// TwinCAT 3 PLC project Coffee_maker_PLC
// ProgramVersion: 3.1.4024.0
// libraries:
//   Tc2_Standard, * (Beckhoff Automation GmbH)
//   Tc2_System, * (Beckhoff Automation GmbH)
//   Tc3_Module, * (Beckhoff Automation GmbH)
// project tree:
//   / GlobalTextList.TcGTLO, PlcTask.TcTTO, Visualization Manager.TcVMO (not stored)
//   GVLs/ GVL.TcGVL
//   POUs/ Cleaning.TcPOU, Fill_Cup.TcPOU, Heat_Water.TcPOU, Lamp_Loop.TcPOU, MAIN.TcPOU, Prepare_Ingredients.TcPOU, Show_Strength.TcPOU
//   VISUs/ Visualization.TcVIS
// real-time tasks:
//   TASK PlcTask: cycle T#10ms, priority 20, ADS port 350
//   TASK Fill_Cup: cycle T#10ms, priority 1, ADS port 351
//   TASK Prepare_Ingredients: cycle T#5ms, priority 2, ADS port 352
//   TASK Heating: cycle T#1ms, priority 3, ADS port 353
//   TASK LoopLamp: cycle T#10ms, priority 4, ADS port 354
//   TASK Show strength: cycle T#10ms, priority 5, ADS port 355

CONFIGURATION Coffee_maker_PLC
    RESOURCE PLC ON TwinCAT3
        TASK PlcTask(INTERVAL := T#10ms, PRIORITY := 20);
        PROGRAM MAIN WITH PlcTask : MAIN;
        PROGRAM Fill_Cup WITH PlcTask : Fill_Cup;
        PROGRAM Heat_Water WITH PlcTask : Heat_Water;
        PROGRAM Lamp_Loop WITH PlcTask : Lamp_Loop;
        PROGRAM Prepare_Ingredients WITH PlcTask : Prepare_Ingredients;
        PROGRAM Show_Strength WITH PlcTask : Show_Strength;
    END_RESOURCE
END_CONFIGURATION

// ---- GVLs/GVL.TcGVL
{attribute 'qualified_only'}
VAR_GLOBAL
	Start : BOOL := FALSE;	
	CleanMachine : BOOL := FALSE;
	FillCup : BOOL := FALSE;
	Water_Warm: BOOL := FALSE;
    Ingredients_Ready : BOOL := FALSE;
	Cup_filled : BOOL := FALSE;
	Coffee_Strength : INT;
	LamploopOn : BOOL := FALSE;
	Strength : INT := 0;
	Lamp1 : BOOL := FALSE; // Output for Lamp 1
    Lamp2 : BOOL := FALSE; // Output for Lamp 2
    Lamp3 : BOOL := FALSE; // Output for Lamp 3
	ShowStrength : BOOL := FALSE;
END_VAR

// ---- POUs/MAIN.TcPOU
PROGRAM MAIN
VAR
	cleaningfb1: Cleaning;
END_VAR

IF gvl.CleanMachine = TRUE THEN 
	Cleaning(TypeCleaning := 1);
END_IF

END_PROGRAM

// ---- POUs/Cleaning.TcPOU
FUNCTION_BLOCK Cleaning
VAR_INPUT
	TypeCleaning : INT;
END_VAR
VAR_OUTPUT
END_VAR
VAR
	MachineClean : BOOL := FALSE;
	CleaningStep : INT := 0;
	WaitTime : TIME := T#2S; // Stel de wachttijd in voor elke stap
    Timer : TIME := T#0s;
    CleaningDone : BOOL := FALSE;
END_VAR

IF TypeCleaning = 1 THEN 
	// grote schoonmaak 
	// Reset schoonmaak gereed status
	MachineClean := FALSE;
	
	IF NOT CleaningDone THEN
		CASE CleaningStep OF
		0:
			// Stap 1: Begin het schoonmaakproces
			Timer := Timer + T#100MS;
			IF Timer >= WaitTime THEN
				CleaningStep := CleaningStep + 1;
				Timer := T#0S; // Reset de timer
			END_IF

		1:
			// Stap 2: Spoel de koffieresiduen uit
			Timer := Timer + T#100MS;
			IF Timer >= WaitTime THEN
				CleaningStep := CleaningStep + 1;
				Timer := T#0S;
			END_IF

		2:
			// Stap 3: Reinig waterleidingen
			Timer := Timer + T#100MS;
			IF Timer >= WaitTime THEN
				CleaningStep := CleaningStep + 1;
				Timer := T#0S;
			END_IF
	
		3:
			// Stap 4: Reinig koffiedikopvangbak
			Timer := Timer + T#100MS;
			IF Timer >= WaitTime THEN
				CleaningStep := CleaningStep + 1;
				Timer := T#0S;
			END_IF

		4:
			// Stap 5: Reinig externe oppervlakken
			Timer := Timer + T#100MS;
			IF Timer >= WaitTime THEN
				CleaningDone := TRUE;  // Schoonmaak is gereed
			END_IF
		ELSE
		// Schoonmaakproces voltooid, zet de returnwaarde op TRUE
		MachineClean := TRUE;
		END_CASE
	END_IF

	
	
ELSIF TypeCleaning = 2 THEN 
	// kleine reineging 
	// Reset schoonmaak gereed status
	MachineClean := FALSE;
	
	
	
	IF NOT CleaningDone THEN
		CASE CleaningStep OF
			0:
				// Stap 1: Spoel koffieresiduen kort door
				Timer := Timer + T#100MS;
				IF Timer >= WaitTime THEN
					CleaningStep := CleaningStep + 1;
					Timer := T#0S; // Reset de timer
				END_IF
	
			1:
				// Stap 2: Spoel waterleidingen kort door
				Timer := Timer + T#100MS;
				IF Timer >= WaitTime THEN
					CleaningStep := CleaningStep + 1;
					Timer := T#0S;
				END_IF
	
			2:
				// Stap 3: Reinig opvangbak oppervlakkig
				Timer := Timer + T#100MS;
				IF Timer >= WaitTime THEN
					CleaningDone := TRUE;  // Kleine schoonmaak is gereed
				END_IF
		ELSE
			// Schoonmaakproces voltooid, zet de returnwaarde op TRUE
			MachineClean := TRUE;
		END_CASE
	END_IF
END_IF

END_FUNCTION_BLOCK

// ---- POUs/Fill_Cup.TcPOU
PROGRAM Fill_Cup
VAR
	Filling : BOOL := FALSE;
	Timer : Ton;
	Licht : BOOL;
	Medium : BOOL; 
	Sterk : BOOL;	
	cleaningfb: Cleaning;
END_VAR

IF gvl.FillCup THEN 
	IF gvl.Water_Warm = TRUE AND gvl.Ingredients_Ready = TRUE THEN
	Timer(IN := TRUE, PT := T#5S); // 5 seconden timer

		IF gvl.Strength = 0 THEN;
			gvl.LamploopOn := true;		
				IF licht  THEN
				gvl.Strength := 1;
				gvl.LamploopOn := FALSE;
				
				ELSIF medium THEN 
				gvl.Strength := 2;
				gvl.LamploopOn := FALSE;
				
				ELSIF sterk THEN
				gvl.Strength := 3;
				gvl.LamploopOn := FALSE;
				END_IF
		END_IF
	
		IF gvl.Strength > 0 THEN
			Filling := TRUE;
			gvl.ShowStrength := 1;
		END_IF
		
		IF Timer.Q THEN 
			Filling := FALSE;
			gvl.Cup_Filled := TRUE;
		END_IF	
		
		Cleaning(TypeCleaning := 2); // korte reiniging 
		
	END_IF
END_IF

END_PROGRAM

// ---- POUs/Heat_Water.TcPOU
PROGRAM Heat_Water
VAR
	WaterTemp: INT := 20;
	Heating : bool := false;
	ELSIFgvl: INT;
	Timer:TON;
	
END_VAR

IF gvl.Start AND WaterTemp <= 85 THEN
    Timer(IN := TRUE, PT := T#100MS);  
    Heating := TRUE;

    IF Timer.Q THEN 
        WaterTemp := WaterTemp + 1;  // Verhoog de temperatuur met 1 graad per seconde
        Timer(IN := FALSE);          // Reset de timer na een seconde
    END_IF

ELSIF gvl.Start = FALSE THEN
    Heating := FALSE;
    Timer(IN := FALSE);              // Zorg ervoor dat de timer wordt gereset als Start FALSE is

ELSIF WaterTemp >= 85 THEN  
    Heating := FALSE;
    gvl.Water_Warm := TRUE;	
    Timer(IN := FALSE);              // Stop de timer als de gewenste temperatuur is bereikt

END_IF

END_PROGRAM

// ---- POUs/Lamp_Loop.TcPOU
PROGRAM Lamp_Loop
VAR
	Strength : INT;
	Lamp1 : BOOL := FALSE; // Output for Lamp 1
    Lamp2 : BOOL := FALSE; // Output for Lamp 2
    Lamp3 : BOOL := FALSE; // Output for Lamp 3

    tCycleTimer : TON; // Timer for cycle timing
    nCycleStep : INT := 0; // State variable to track which lamp is on 
END_VAR

IF gvl.LamploopOn THEN 
	// Timer instellingen
	tCycleTimer(IN := TRUE, PT := T#0.5S); // De timer is ingesteld op 2 seconden
	
	IF tCycleTimer.Q THEN
		tCycleTimer(IN := FALSE);  // Stop de timer zodra deze is afgelopen
		tCycleTimer(IN := TRUE);   // Reset de timer voor de volgende cyclus
	
		// Volgende stap van de cyclus
		nCycleStep := nCycleStep + 1;
		
		IF nCycleStep > 2 THEN
			nCycleStep := 0; // Reset de cyclus na 3 stappen
		END_IF
	END_IF
	
	// Lamp logica
	CASE nCycleStep OF
		0: // Lamp 1 aan, andere uit
			gvl.Lamp1 := TRUE;
			gvl.Lamp2 := FALSE;
			gvl.Lamp3 := FALSE;
		1: // Lamp 2 aan, andere uit
			gvl.Lamp1 := FALSE;
			gvl.Lamp2 := TRUE;
			gvl.Lamp3 := FALSE;
		2: // Lamp 3 aan, andere uit
			gvl.Lamp1 := FALSE;
			gvl.Lamp2 := FALSE;
			gvl.Lamp3 := TRUE;
	END_CASE
END_IF

END_PROGRAM

// ---- POUs/Prepare_Ingredients.TcPOU
PROGRAM Prepare_Ingredients
VAR
	BoneContainer: REAL := 0;	
	Prepairing : BOOL := FALSE;
	Timer:TON;
END_VAR

Timer(IN := TRUE, PT := T#100MS); 				// 1 seconden timer

IF gvl.Start AND BoneContainer <= 90 THEN
    Timer(IN := TRUE, PT := T#1S);   		// Stel de timer in om elke seconde af te gaan
    Prepairing := TRUE;

    IF Timer.Q THEN
        BoneContainer := BoneContainer + 1;  // Verhoog de inhoud van BoneContainer met 1
        Timer(IN := FALSE);                  // Reset de timer na een seconde
    END_IF

ELSIF BoneContainer >= 90 THEN
    gvl.Ingredients_Ready := TRUE;
    Prepairing := FALSE;
    Timer(IN := FALSE);                      // Stop de timer wanneer BoneContainer vol is

ELSIF gvl.Start = FALSE THEN
    Prepairing := FALSE;
    Timer(IN := FALSE);                      // Reset de timer wanneer Start FALSE is
END_IF

END_PROGRAM

// ---- POUs/Show_Strength.TcPOU
PROGRAM Show_Strength
VAR
END_VAR

IF gvl.ShowStrength = TRUE THEN 
	gvl.lamp1 := 0;
	gvl.Lamp2 := 0;
	gvl.Lamp3 := 0;
	
	IF gvl.Strength = 1 THEN 
		gvl.Lamp1 := 1;
	ELSIF gvl.Strength = 2 THEN 
		gvl.Lamp2 := 1;
	ELSIF gvl.Strength = 3 THEN 
		gvl.Lamp3 := 1;
	END_IF
	gvl.ShowStrength := 0;
	
END_IF

END_PROGRAM

// ---- GlobalTextList.TcGTLO
TEXTLIST GlobalTextList
  313 = 'Cleaning Program'
  896 = 'Filling Cup'
  750 = 'Heating'
  77 = 'Koffie klaar'
  777 = 'Licht          Medium        Sterk'
  759 = 'Prepairing Ingredients'
  169 = 'Start'
  681 = 'Start Cleaning Program'
  172 = 'Watertemperatuur'
END_TEXTLIST

// ---- VISUs/Visualization.TcVIS
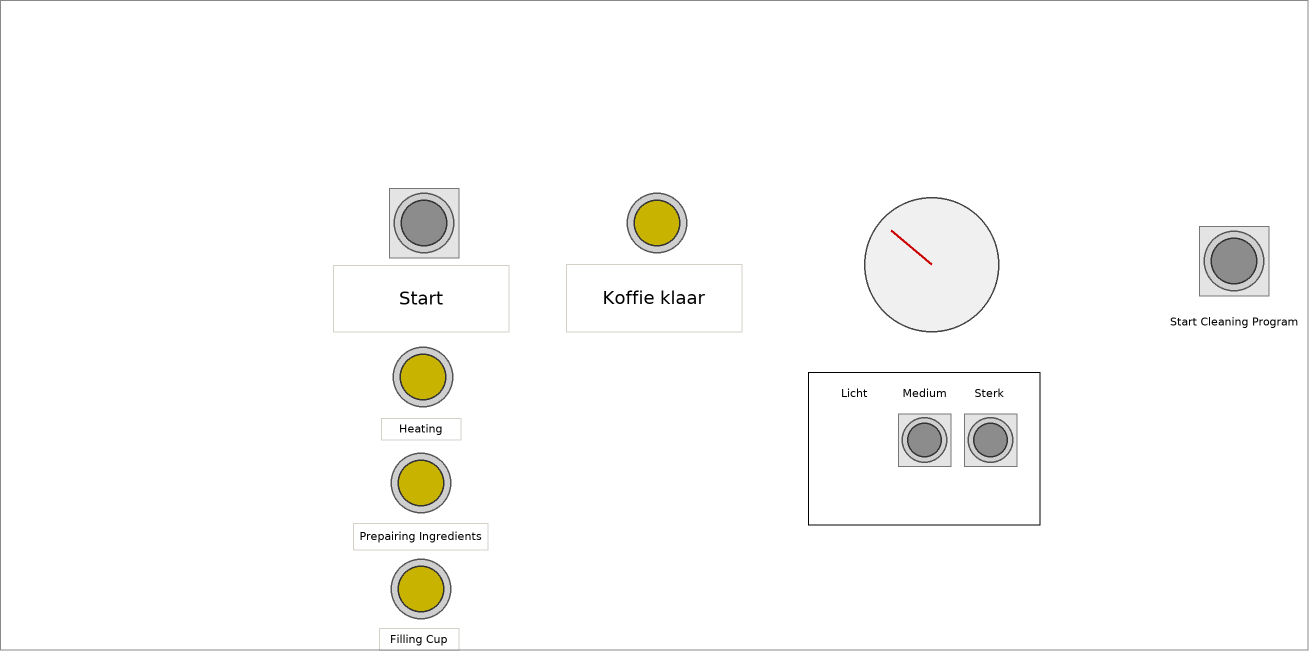
VISUALIZATION Visualization  // 1309x651
    Lamp1 (388,342 70x70), variable: Heating.Heating, style: Lamp-Lamp1-Yellow
    Lamp1 (386,448 70x70), variable: Prepare_Ingredients.Prepairing, style: Lamp-Lamp1-Yellow
    PushSwitchLed (389,188 70x70), variable: GVL.Start, behaviour: TOGGLE, style: Switch-PushSwitchLed-Gray
    Textfield (333,265 176x67), "Start"
    Textfield (381,418 80x22), "Heating"
    Textfield (353,523 135x27), "Prepairing Ingredients"
    Lamp1 (622,188 70x70), variable: Fill_Cup.Ready, style: Lamp-Lamp1-Yellow
    Textfield (566,264 176x68), "Koffie klaar"
    Meter180 (788,197 287x135), value: Heating.WaterTemp, style: Meter-Meter180-Yellow, scale format: %.1f, scale 0..100
        p518627256: Watertemperatuur
    Lamp1 (386,554 70x70), variable: Fill_Cup.Filling, style: Lamp-Lamp1-Yellow
    Textfield (379,628 80x23), "Filling Cup"
    Lamp1 (840,473 41x38), variable: Lamp_Loop.Lamp1, style: Lamp-Lamp1-Yellow
    Lamp1 (907,473 41x38), variable: Lamp_Loop.Lamp2, style: Lamp-Lamp1-Yellow
    Lamp1 (972,473 41x38), variable: Lamp_Loop.Lamp3, style: Lamp-Lamp1-Yellow
    Frame (979,444 1x0)
    PushSwitch (832,410 53x60), variable: Fill_Cup.Licht, behaviour: TOGGLE, style: Switch-PushSwitch-Gray
    Rectangle (808,372 232x153)
    Textfield (813,378 219x31), "Licht Medium Sterk"
    PushSwitch (898,410 53x60), variable: Fill_Cup.Medium, behaviour: TOGGLE, style: Switch-PushSwitch-Gray
    PushSwitch (964,410 53x60), variable: Fill_Cup.Sterk, behaviour: TOGGLE, style: Switch-PushSwitch-Gray
    PushSwitch (1199,226 70x70), variable: GVL.CleanMachine, behaviour: TOGGLE, style: Switch-PushSwitch-Gray
    Label (1159,307 150x30), "Start Cleaning Program"
END_VISUALIZATION
